// TIA Portal V19 export
VAR_GLOBAL   // PLC tag table "Default tag table"
   Tag_1 AT %T1 : Timer;
END_VAR
